TYPE "FeedMachine_Par"
VERSION : 0.1
// Block: FeedMachine_Par
   STRUCT
      Man : Struct
         VelBwd : LReal;
         VelFwdHigh : LReal;
         VelFwdLow : LReal;
         Acc : LReal;
         Dec : LReal;
         Jerk : LReal;
         DelayChangeVel : Time;
      END_STRUCT;
   END_STRUCT;

END_TYPE
